// SIMATIC S7-200 project (STEP 7-Micro/WIN), CPU 224XP REL 02.01

SYMBOL_TABLE USR1
Always_On        SM0.0    // This bit is always on.
First_Scan_On    SM0.1    // This bit is on for the first scan cycle only.
Time_0_Intrvl    SMB34    // Specifies time interval (in 1-ms increments from 5 to 255): timed interrupt 0.
HSC1_Ctrl        SMB47    // This byte enables you to control the operation of high-speed counter 1.
HSC1_CV          SMD48    // New current value of high-speed counter 1. SMB48 is the most significant byte.
HSC1_PV          SMD52    // New preset value of high-speed counter 1. SMB52 is the most significant byte.
Display_Voltage  QB0      // LEDs attached to this output display the voltage value.
END_SYMBOL_TABLE

ORGANIZATION_BLOCK MAIN:OB1
TITLE=
//  题目：
//  用S7-200 CPU 214的高速计数器HSC累计来自模拟量/频率转换器(A/F)的脉冲来模拟电压值
// ***概述***
// 本例说明了如何利用CPU 214的高速计数器HSC及频率转换器来计算模拟电压。首先频率转换
// 器将输入电压(0-10V)转换为矩形脉冲信号(0-2000Hz)，再将此信号送入CPU 214高速记数器
// 的输入端并累计脉冲数。当预置的间隔时间到后，通过累计脉冲数，计算出被测模拟电压值。
// 硬件要求
// 需要使用如下设备：
// 1台   CPU214          AC/AD/RLY或DC/DC/DC
// 1台  电压/频率转换器      SFW01(Trankner　Company)
// (地址：Engineering Office Trankner, Industrial Area North PF38,09618 Brand-Erbisdort,
// Germany)
// 计数参数：      供电电压      24V DC
//                 输入          0-10v DC
//                 输出          方波，GND-24V
//                 测量范围      0-10V 0-2000Hz
//                 比率          200Hz/V (线性)
// ***程序结构***
// 
//  主程序	在第一个扫描周期调用子程序SBR0
//  SBR0	高速计数器和定时中断的初始化
//  INT0	对高速计数器求值的定时中断程序
// 
// 
// ***程序和注释***
// 主程序在第一个扫描周期调用初始化程序SBR0,仅在第一个扫描周期标志位SM0.1=1
// 由子程序实现初始化。首先，把高速计数器HSC1的控制字节SMB47置为16进制数'FC'
// 其含义是：正方向计数，可更新预置值(PV)，可更新当前值(CV),激活HSC1
// 然后，用指令'HDEF'把高速计数器HSC1置成工作模式0，即没有复位或起始输入，也没有
// 外部的方向选择。当前值SMD48复位为0预置值SMD52置为FFFF(十六进制).定时中断0间隔
// 时间SMB34置为100ms,中断程序0分配给定时中断0(中断事件10),并允许中断。用指
// 令HSC1启动高速计数器。
// 每100ms调用一次中断程序0，读出高速计数器的数值后将其置零。通过HSC1计数值及变换
// 关系(0-2kHz对应于0-10V)来求被测的模拟电压值。本例中，计数值仅除以2，然后置入输
// 出字节QB0,以便通过LED来显示被测的电压值。显示值与10倍真实电压值相对应。例如，
// 计数值为200除以2是100，那么被测的模拟电压值就是10.0V。因为计数器100ms内共有200
// 个计数脉冲，这正与2000Hz-10V相对应， 假设计数值为104，则实际电压值应为5.2V
// 注意：定时中断间隔时间可在5-255ms的范围内变化，然而通过设立一个标志，可根据需要
// 来延长高速计数器的求值和复位时间，这样就有更长的扫描间隔，以便提高精确度，同时
// 也会带来更长的更新时间。例如，定时中断设为100ms,每调用一次，标志增加1，仅当标志
// 满10时，才对高速计数器求值和复位。也就是说，10V电压可接收的最大脉冲为2000，这
// 样，求值精确到5/1000V,即精确度是上例的10倍，但同时速度也减慢了10倍。
// 
// 
BEGIN
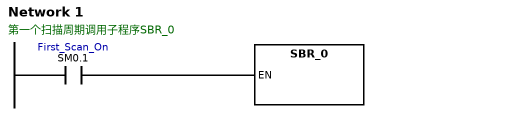
Network 1 // 	
// 第一个扫描周期调用子程序SBR_0
// 仅首次扫描时，SM0.1=1
// 调用子程序0
LD     First_Scan_On:SM0.1
CALL   SBR_0:SBR0
Network 2 //  主程序结束.
// MEND				
// 
// 
// 
Network 3 // ***子程序0***
// 
// 
// 
Network 4 //  //***中断程序0***
//  Start INT0.
// 
END_ORGANIZATION_BLOCK

SUBROUTINE_BLOCK SBR_0:SBR0
TITLE=
BEGIN
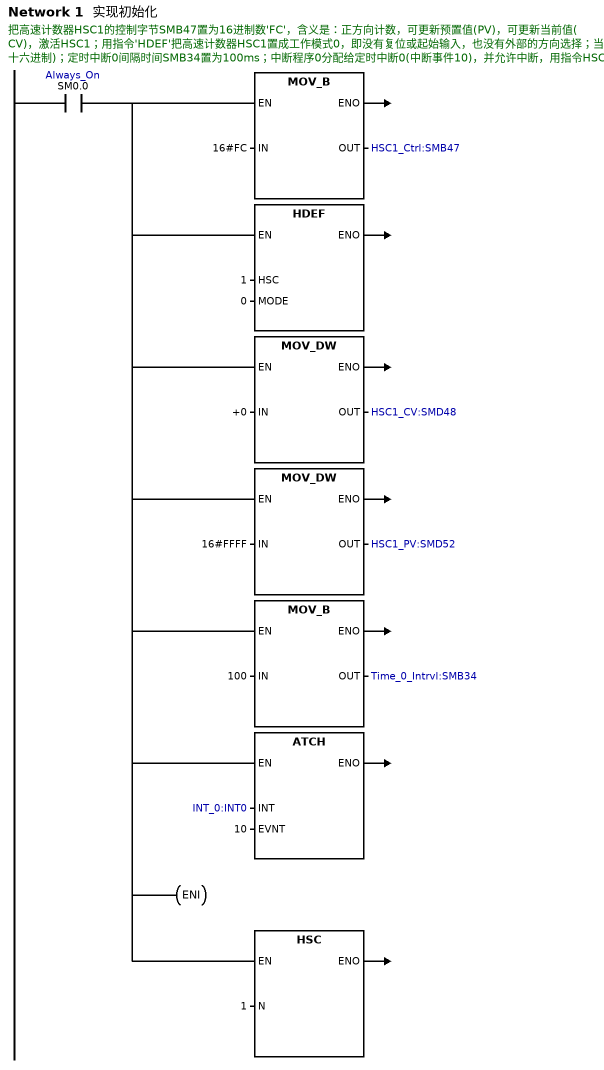
Network 1 // 实现初始化
// 把高速计数器HSC1的控制字节SMB47置为16进制数'FC'，含义是：正方向计数，可更新预置值(PV)，可更新当前值(CV)，激活HSC1；用指令'HDEF'把高速计数器HSC1置成工作模式0，即没有复位或起始输入，也没有外部的方向选择；当前值SMD48复位为0，预置值SMD52置为FFFF(十六进制)；定时中断0间隔时间SMB34置为100ms；中断程序0分配给定时中断0(中断事件10)，并允许中断，用指令HSC1启动高速计数器
// SM0.0总是1
// 设置HSC1控制字节：上升沿复位，上升沿起动，
// 1*计数速率，正向计数，可改变方向，可更新PV,
// 可更新CV(当前值),激活HSC1
// HSC1工作于模式0
// HSC1当前值复位
// 设置HSC1预置值，（本例未用）
// 设置定时中断0间隔时间为100ms
// 指定定时中断事件10 调用中断程序0
// 允许所有中断
// 起动高速计数器 HSC1.
LD     Always_On:SM0.0
MOVB   16#FC, HSC1_Ctrl:SMB47
HDEF   1, 0
MOVD   +0, HSC1_CV:SMD48
MOVD   16#FFFF, HSC1_PV:SMD52
MOVB   100, Time_0_Intrvl:SMB34
ATCH   INT_0:INT0, 10
ENI
HSC    1
Network 2 //  子程序0结束
// RET					
// 
END_SUBROUTINE_BLOCK

INTERRUPT_BLOCK INT_0:INT0
TITLE=
BEGIN
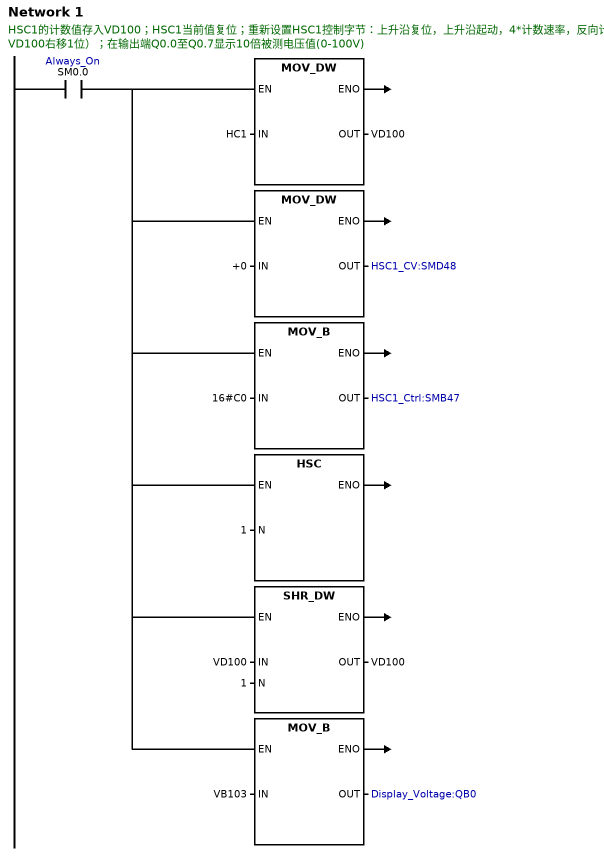
Network 1
// HSC1的计数值存入VD100；HSC1当前值复位；重新设置HSC1控制字节：上升沿复位，上升沿起动，4*计数速率，反向计数，不改变方向不更新PV，可更新CV，激活HSC1；启动高速计数器HSC1；SC1的计数值除以2（即VD100右移1位）；在输出端Q0.0至Q0.7显示10倍被测电压值(0-100V)
// SM0.0总是1.
// HSC1的计数值存入VD100
// HSC1当前值复位，
// 重新设置HSC1控制字节：上升沿复位，上升
// 沿起动，4*计数速率，反向计数，不改变方向
// 不更新PV,可更新CV，激活HSC1
// 起动高速计数器，HSC1
// HSC1的计数值除以2（即VD100右移1位）
// 在输出端Q0.0至Q0.7显示10倍被测电压值(0-100V)
LD     Always_On:SM0.0
MOVD   HC1, VD100
MOVD   +0, HSC1_CV:SMD48
MOVB   16#C0, HSC1_Ctrl:SMB47
HSC    1
SRD    VD100, 1
MOVB   VB103, Display_Voltage:QB0
Network 2 // 结束中断程序0
// RETI					
// 
END_INTERRUPT_BLOCK
